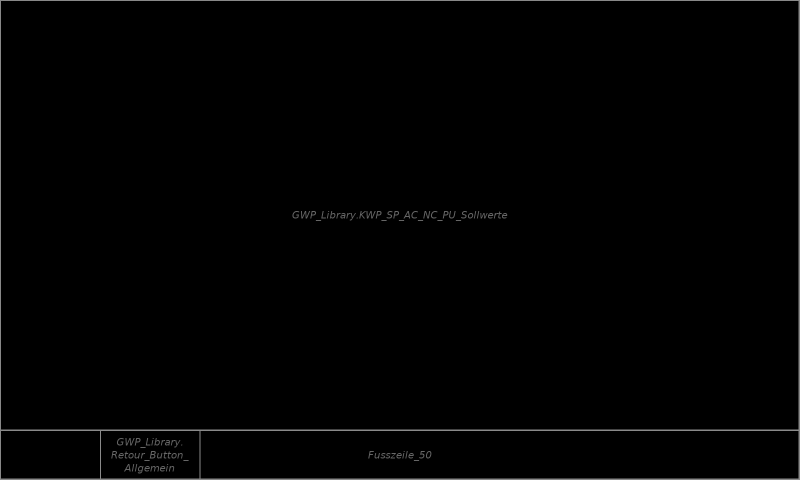
VISUALIZATION KWP_SP_AC_NC_PU_Sollwerte  // 800x480
    Frame (0,0 800x430)
        shows GWP_Library.KWP_SP_AC_NC_PU_Sollwerte(FB_KWP_SP_AC_NC := Main.KWP_SP_AC_NC_0)
    Frame (0,430 800x50)
        shows Fusszeile_50()
    Frame (100,430 100x50)
        shows GWP_Library.Retour_Button_Allgemein()
END_VISUALIZATION

(* stored: Version 1.1.0.1, ProductVersion 3.1.4022.6
   Visu KWP_SP_AC_NC_PU_Sollwerte: Id {f311845f-d1b1-4936-af2f-1f63b3a5f1fd} *)
